FUNCTION_BLOCK PTRC (* Composite Function Block Type *)
  (* Standard: 61499-2 *)
  (* Version 0.0, 12/10/2023, Cheyan, Schneider Electric, template *)
  PACKAGE Main;
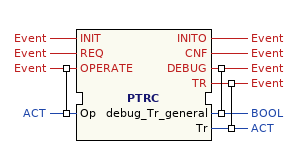
  EVENT_INPUT
    INIT; (* Initialization Request *)
    REQ; (* Normal Execution Request *)
    OPERATE WITH Op;
  END_EVENT
  EVENT_OUTPUT
    INITO; (* Initialization Confirm *)
    CNF; (* Execution Confirmation *)
    DEBUG WITH debug_Tr_general;
    TR WITH Tr;
  END_EVENT
  VAR_INPUT
    Op : ACT; (* Input event qualifier *)
  END_VAR
  VAR_OUTPUT
    debug_Tr_general : BOOL;
    Tr : ACT; (* Output event qualifier *)
  END_VAR
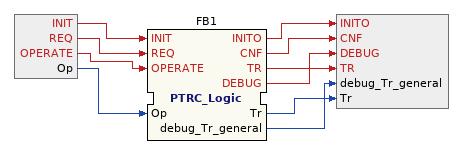
  FBS
    FB1 : PTRC_Logic;
  END_FBS
  EVENT_CONNECTIONS
    FB1.INITO TO INITO;
    FB1.CNF TO CNF;
    INIT TO FB1.INIT;
    REQ TO FB1.REQ;
    FB1.DEBUG TO DEBUG;
    OPERATE TO FB1.OPERATE;
    FB1.TR TO TR;
  END_CONNECTIONS
  DATA_CONNECTIONS
    FB1.debug_Tr_general TO debug_Tr_general;
    Op TO FB1.Op;
    FB1.Tr TO Tr;
  END_CONNECTIONS
END_FUNCTION_BLOCK
